// TwinCAT 3 PLC project HD_PLC
// ProgramVersion: 3.1.4024.0
// libraries:
//   Tc2_ModbusRTU, * (Beckhoff Automation GmbH)
//   Tc2_Standard, * (Beckhoff Automation GmbH)
//   Tc2_System, * (Beckhoff Automation GmbH)
//   Tc2_Utilities, * (Beckhoff Automation GmbH)
//   Tc3_Module, * (Beckhoff Automation GmbH)
//   VisuDialogs, * (System)
//   VisuSymbols,3.5.10.0,System
// project tree:
//   / GlobalTextList.TcGTLO, PlcTask.TcTTO, Visualization Manager.TcVMO (not stored), VISU_TASK.TcTTO
//   GVLs/ HMI_Global.TcGVL
//   POUs/ MAIN.TcPOU, SYSTEM.TcPOU
//   VISUs/ Data_Left.TcVIS, Footer.TcVIS, Header.TcVIS, Header_2.TcVIS, ImagePool.TcIPO (not stored), MainScreen.TcVIS, RinseMode.TcVIS, RinseMode_Footer.TcVIS, Set.TcVIS, Set_Output.TcVIS, Set_Input.TcVIS, Set_Sensor.TcVIS, Visualization.TcVIS
// real-time tasks:
//   TASK PlcTask: cycle T#10ms, priority 20, ADS port 350
//   TASK VISU_TASK: cycle T#10ms, priority 1, ADS port 351
//   TASK VISU_TASK1: cycle T#200000us, priority 30, ADS port 352

CONFIGURATION HD_PLC
    RESOURCE PLC ON TwinCAT3
        TASK PlcTask(INTERVAL := T#10ms, PRIORITY := 20);
        TASK VISU_TASK(INTERVAL := T#200000us, PRIORITY := 30);
        PROGRAM MAIN WITH PlcTask : MAIN;
        PROGRAM SYSTEM WITH PlcTask : SYSTEM;
        PROGRAM VisuElems_Visu_Prg WITH VISU_TASK : VisuElems.Visu_Prg;
    END_RESOURCE
END_CONFIGURATION

// ---- GVLs/HMI_Global.TcGVL
{attribute 'qualified_only'}
VAR_GLOBAL
	//HMI Stuff
	HMI_OUT_Digital 	: ARRAY[0..31] OF BOOL;
	HMI_OUT_Analog 		: ARRAY[0..31] OF INT;
	
	HMI_IN_Digital 		: ARRAY[0..31] OF BOOL;
	HMI_IN_Analog 		: ARRAY[0..31] OF INT;
	
	HMI_IN_Temp 		: ARRAY[0..4] OF REAL;
	
	HMI_State			: INT;
	
	fbGetLocalSystemTime: FB_LocalSystemTime;
	sSystemDateTime : STRING;
	sSystemTime		: STRING;
	sSystemDate		: STRING;
	
	HMI_ArrayGraph1 : ARRAY[0..1] OF INT;
	HMI_ArrayGraph2 : ARRAY[0..1] OF INT;
	HMI_ArrayGraph3 : ARRAY[0..1] OF INT;

END_VAR

// ---- POUs/MAIN.TcPOU
PROGRAM MAIN
VAR
	
	CountScale : BYTE;

	Mux_Select AT %Q*: ARRAY[0..4] OF BOOL;	
	ADC_Val AT %I* : INT; 
	AnalogRead : ARRAY[0..31] OF INT;
	CLK_MUX : BOOL;
	
	MUX_FUNC : MUX_ADC;

	IO_Out AT %Q* : ARRAY[0..31] OF BOOL;
	IO_In AT %I* : ARRAY[0..16] OF BOOL;
	
	SensAnalaog AT %I* : ARRAY[0..3] OF INT;
	
	RTD_ADC AT %I* : INT;
	RTD_Temp : REAL;
	
	

END_VAR

CLK_MUX := NOT(CLK_MUX);

IO_Out[8] := HMI_Global.HMI_IN_Digital[0];
HMI_Global.HMI_OUT_Analog[0] := AnalogRead[9];

IF AnalogRead[9] > 1000 THEN
	HMI_Global.HMI_OUT_Digital[0] := TRUE;
ELSE
	HMI_Global.HMI_OUT_Digital[0] := FALSE;
END_IF
 

MUX_FUNC(
	CLK := CLK_MUX,
	ADC_INPUT := ADC_Val,
	SELLECT => Mux_Select,
	ADC_OUTPUT => AnalogRead	
);

END_PROGRAM

// ---- POUs/SYSTEM.TcPOU
PROGRAM SYSTEM
VAR
END_VAR

HMI_Global.fbGetLocalSystemTime(
	sNetID:= , 
	bEnable:= TRUE, 
	dwCycle:= 1, 
	dwOpt:= , 
	tTimeout:= , 
	bValid=> , 
	systemTime=> , 
	tzID=> );
	
HMI_Global.sSystemDateTime := SYSTEMTIME_TO_STRING(HMI_Global.fbGetLocalSystemTime.systemTime);
HMI_Global.sSystemDate := MID(STR:= HMI_Global.sSystemDateTime, LEN:=10, POS:=1);
HMI_Global.sSystemTime := MID(STR:= HMI_Global.sSystemDateTime, LEN:=8, POS:=12);

END_PROGRAM

// ---- GlobalTextList.TcGTLO
TEXTLIST GlobalTextList
  734 = '%1.1f'
  899 = '%2.2f'
  70 = '%i'
  841 = '%s'
  97 = '10'
  56 = '120'
  900 = '30'
  405 = '36'
  563 = '60'
  451 = 'A. PRESS'
  564 = 'B1'
  765 = 'B10'
  285 = 'B11'
  111 = 'B12'
  897 = 'B13'
  671 = 'B14'
  804 = 'B15'
  328 = 'B16'
  300 = 'B17'
  486 = 'B18'
  957 = 'B19'
  273 = 'B2'
  588 = 'B20'
  314 = 'B21'
  91 = 'B22'
  991 = 'B23'
  768 = 'B24'
  634 = 'B25'
  160 = 'B26'
  185 = 'B27'
  572 = 'B28'
  78 = 'B29'
  783 = 'B3'
  964 = 'B30'
  98 = 'B31'
  326 = 'B32'
  703 = 'B4'
  227 = 'B5'
  844 = 'B6'
  235 = 'B7'
  599 = 'B8'
  248 = 'B9'
  100 = 'BACK'
  372 = 'Bic.'
  816 = 'BLOOD PUMP'
  325 = 'Button 1'
  42 = 'Button 2'
  879 = 'Button 3'
  476 = 'Button 4'
  556 = 'Button 5'
  421 = 'Button 6'
  73 = 'Button 7'
  541 = 'Button 8'
  424 = 'Button 9'
  46 = 'BY PAS'
  570 = 'BYPASS'
  2 = 'BYPASS\nRELEASE'
  359 = 'CHECK AND TEST FUNCTION'
  724 = 'CONC. SET'
  918 = 'COND.'
  942 = 'D. PRESS'
  223 = 'DIALYSE'
  633 = 'DIALYSIS'
  645 = 'EST. UF TIME'
  400 = 'HEMODIALYSIS'
  102 = 'HMI STATE'
  583 = 'INPUT'
  17 = 'Input'
  280 = 'Input \nDigital'
  439 = 'Input Digital'
  212 = 'InputDigital'
  770 = 'ISO-UF\n[1sec]'
  733 = 'mmHg'
  339 = 'Na'
  358 = 'NEXT'
  851 = 'ON / OFF'
  71 = 'OUTPUT'
  279 = 'PREP'
  48 = 'PREP. COMP.'
  59 = 'PRIM.'
  370 = 'RINSE\nMODE'
  863 = 'S/N\n[1sec]'
  925 = 'SENSOR'
  498 = 'SET'
  446 = 'TEMP.'
  666 = 'Temperature'
  237 = 'TEST'
  818 = 'UF DATA'
  819 = 'UF FINISH TIME'
  812 = 'UF GOAL'
  795 = 'UF RATE'
  493 = 'UF REMOVED'
  45 = 'V. PRESS'
  944 = '[C]'
  752 = '[h:min]'
  79 = '[L/h]'
  193 = '[L]'
  495 = '[mEq/L]'
  6 = '[mL/min]'
  374 = '[mS/cm]'
END_TEXTLIST

// ---- VISUs/Data_Left.TcVIS
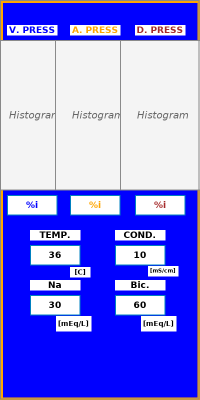
VISUALIZATION Data_Left  // 200x400
    Rectangle (0,0 200x400)
    Histogram (-8,40 86x150), scale format: %1.1f, scale -100..300
        p518627256: mmHg
        p1518820177: HMI_Global.HMI_ArrayGraph1
        p102497268: HMI_Global.HMI_ArrayGraph1
        p788070771: ARRAY [0..1] OF INT
    Histogram (55,40 86x150), scale format: %1.1f, scale -300..100
        p518627256: mmHg
        p1518820177: HMI_Global.HMI_ArrayGraph2
        p102497268: HMI_Global.HMI_ArrayGraph2
        p788070771: ARRAY [0..1] OF INT
    Histogram (120,40 86x150), scale format: %1.1f, scale -400..300
        p518627256: mmHg
        p1518820177: HMI_Global.HMI_ArrayGraph3
        p102497268: HMI_Global.HMI_ArrayGraph3
        p788070771: ARRAY [0..1] OF INT
    Textfield (7,25 50x10), "V. PRESS"
    Textfield (70,25 50x10), "A. PRESS"
    Textfield (135,25 50x10), "D. PRESS"
    Textfield (7,195 50x20), "%i"
    Textfield (70,195 50x20), "%i"
    Textfield (135,195 50x20), "%i"
    Textfield (30,245 50x20), "36"
    Textfield (115,295 50x20), "60"
    Textfield (115,245 50x20), "10"
    Textfield (30,295 50x20), "30"
    Textfield (30,230 50x10), "TEMP."
    Textfield (115,230 50x10), "COND."
    Textfield (115,280 50x10), "Bic."
    Textfield (30,280 50x10), "Na"
    Textfield (70,267 20x10), "[C]"
    Textfield (148,266 30x10), "[mS/cm]"
    Textfield (56,316 35x15), "[mEq/L]"
    Textfield (141,316 35x15), "[mEq/L]"
END_VISUALIZATION

// ---- VISUs/Footer.TcVIS
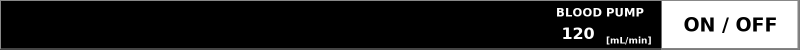
VISUALIZATION Footer  // 800x50
    Rectangle (0,0 800x50)
    Button (661,0 139x50), "ON / OFF"
    Textfield (550,0 100x25), "BLOOD PUMP"
    Textfield (528,21 100x25), "120"
    Textfield (579,28 100x25), "[mL/min]"
END_VISUALIZATION

// ---- VISUs/Header.TcVIS
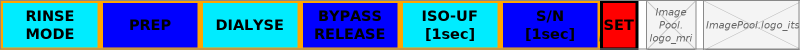
VISUALIZATION Header  // 800x50
    Rectangle (0,0 100x50), "RINSE MODE"
    Rectangle (100,0 100x50), "PREP"
    Rectangle (200,0 100x50), "DIALYSE"
    Rectangle (300,0 100x50), "BYPASS RELEASE", tooltip "BY PAS"
    Rectangle (400,0 100x50), "ISO-UF [1sec]"
    Rectangle (500,0 100x50), "S/N [1sec]"
    Image (600,0 25x50), image: ImagePool.logo_its
    Image (646,0 50x50), image: ImagePool.logo_mri
    Rectangle (600,0 38x50), "SET"
    Image (703,0 100x50), image: ImagePool.logo_its
END_VISUALIZATION

// ---- VISUs/Header_2.TcVIS
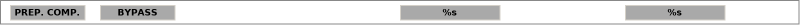
VISUALIZATION Header_2  // 800x25
    Textfield (400,5 75x15), "PREP. COMP."
    Textfield (100,5 75x15), "BYPASS"
    Textfield (400,5 100x15), "%s", text variable: HMI_Global.sSystemDate
    Textfield (625,5 100x15), "%s", text variable: HMI_Global.sSystemTime
    Textfield (10,5 75x15), "PREP. COMP."
END_VISUALIZATION

// ---- VISUs/MainScreen.TcVIS
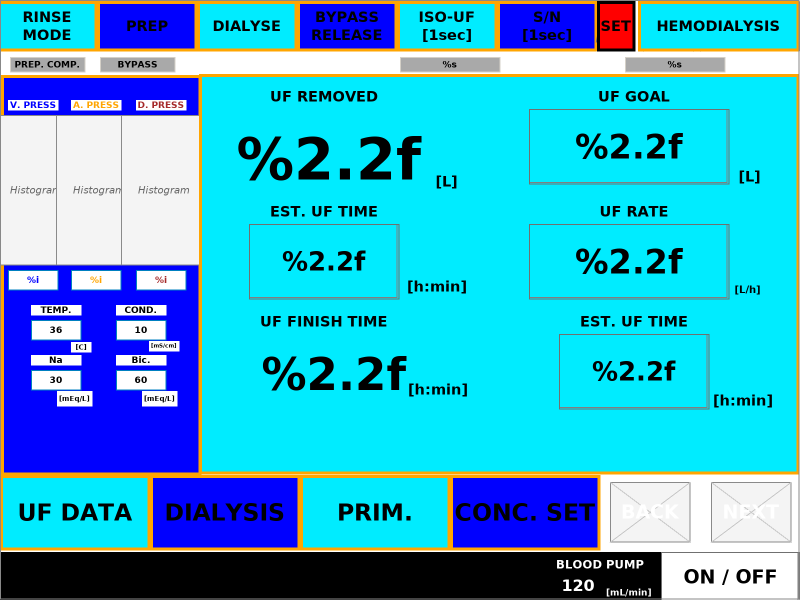
VISUALIZATION MainScreen  // 800x600
    Frame (0,52 800x25)
        shows Header_2()
    Frame (0,552 800x50)
        shows Footer()
    Frame (1,75 200x400)
        shows Data_Left()
    Frame (0,475 800x75)
        shows RinseMode_Footer()
    Rectangle (-3,1 100x50), "RINSE MODE"
        OnMouseClick: FrameSelectionChange Selection=SelectedFrame=2b0ef998-403b-4e78-a897-9d833b853fee, GlobSel=AssignType=Directly, SelType=Locally
    Rectangle (97,1 100x50), "PREP"
    Rectangle (197,1 100x50), "DIALYSE"
    Rectangle (297,1 100x50), "BYPASS RELEASE", tooltip "BY PAS"
    Rectangle (397,1 100x50), "ISO-UF [1sec]"
    Rectangle (497,1 100x50), "S/N [1sec]"
    Image (597,1 25x50), image: ImagePool.logo_its
    Image (643,1 50x50), image: ImagePool.logo_mri
    Rectangle (597,1 38x50), "SET"
        OnMouseClick: FrameSelectionChange Selection=SelectedFrame=2b0ef998-403b-4e78-a897-9d833b853fee, Selection=1, GlobSel=AssignType=Directly, SelType=Locally
    Image (700,1 100x50), image: ImagePool.logo_its
    Frame (199,74 600x400)
        shows RinseMode()
        shows Set()
    Rectangle (638,1 161x50), "HEMODIALYSIS"
END_VISUALIZATION

// ---- VISUs/RinseMode.TcVIS
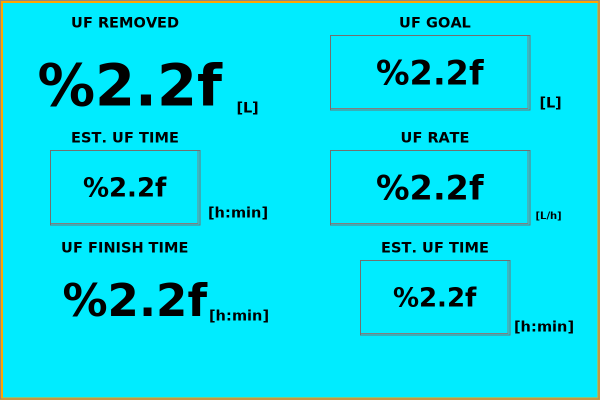
VISUALIZATION RinseMode  // 600x400
    Textfield (0,0 600x400)
    Textfield (50,10 150x25), "UF REMOVED"
    Textfield (360,125 150x25), "UF RATE"
    Textfield (5,35 250x100), "%2.2f"
    Button (330,35 200x75), "%2.2f"
        OnMouseDown: write the text variable via VisuDialogs.Numpad, min 0, max 1000
    Textfield (360,10 150x25), "UF GOAL"
    Button (330,150 200x75), "%2.2f"
        OnMouseDown: write the text variable via VisuDialogs.Numpad, min 0, max 1000
    Button (50,150 150x75), "%2.2f"
        OnMouseDown: write the text variable via VisuDialogs.Numpad, min 0, max 1000
    Textfield (50,125 150x25), "EST. UF TIME"
    Textfield (779,143 1x0)
    Textfield (536,203 25x25), "[L/h]"
    Textfield (538,90 25x25), "[L]"
    Textfield (235,95 25x25), "[L]"
    Textfield (206,200 64x25), "[h:min]"
    Button (360,260 150x75), "%2.2f"
        OnMouseDown: write the text variable via VisuDialogs.Numpad, min 0, max 1000
    Textfield (360,235 150x25), "EST. UF TIME"
    Textfield (512,314 64x25), "[h:min]"
    Textfield (10,250 250x100), "%2.2f"
    Textfield (50,235 150x25), "UF FINISH TIME"
    Textfield (207,303 64x25), "[h:min]"
END_VISUALIZATION

// ---- VISUs/RinseMode_Footer.TcVIS
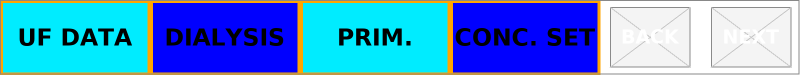
VISUALIZATION RinseMode_Footer  // 800x75
    Textfield (0,0 150x75), "UF DATA"
    Textfield (150,0 150x75), "DIALYSIS"
    Textfield (300,0 150x75), "PRIM."
    Textfield (450,0 150x75), "CONC. SET"
    Image (610,7 80x60), "BACK", image: VisuSymbols.Symbols.ArrowBoldLeft
    Image (711,7 80x60), "NEXT", image: VisuSymbols.Symbols.ArrowBoldRight
END_VISUALIZATION

// ---- VISUs/Set.TcVIS
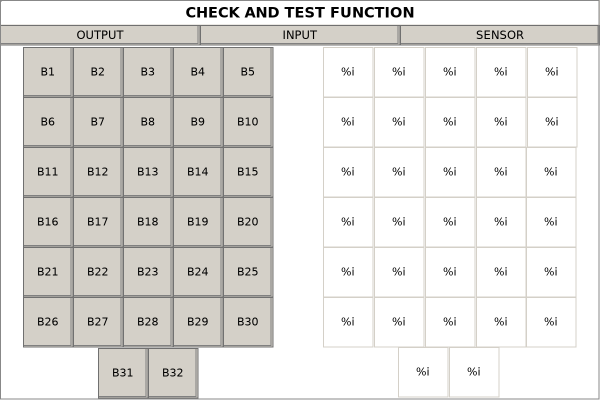
VISUALIZATION Set  // 600x400
    Textfield (0,0 600x25), "CHECK AND TEST FUNCTION"
    Rectangle (0,0 1x0)
    Frame (3,45 600x355)
        shows Set_Output()
        shows Set_Input()
        shows Set_Sensor()
    Button (0,25 200x20), "OUTPUT"
        OnMouseClick: FrameSelectionChange Selection=SelectedFrame=0fef5f47-d526-41e0-bfa2-b91095b14cc7, GlobSel=AssignType=Directly, SelType=Locally
    Button (400,25 200x20), "SENSOR"
        OnMouseClick: FrameSelectionChange Selection=SelectedFrame=0fef5f47-d526-41e0-bfa2-b91095b14cc7, Selection=2, GlobSel=AssignType=Directly, SelType=Locally
    Button (200,25 200x20), "INPUT"
        OnMouseClick: FrameSelectionChange Selection=SelectedFrame=0fef5f47-d526-41e0-bfa2-b91095b14cc7, Selection=1, GlobSel=AssignType=Directly, SelType=Locally
END_VISUALIZATION

// ---- VISUs/Set_Output.TcVIS
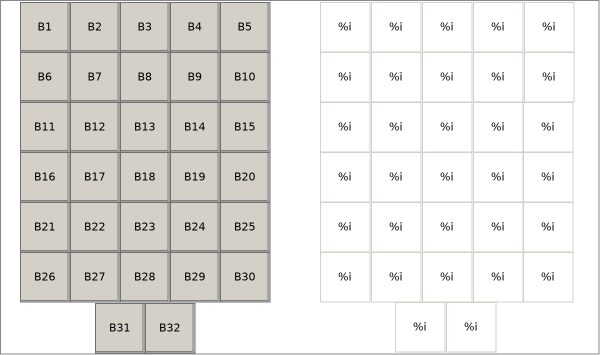
VISUALIZATION Set_Output  // 600x355
    Button (20,2 50x50), "B1", colour toggle: HMI_Global.HMI_OUT_Digital[0]
        toggle HMI_Global.HMI_OUT_Digital[0]
    Textfield (320,2 50x50), "%i", text variable: HMI_Global.HMI_OUT_Analog[0]
        OnMouseDown: write the text variable via VisuDialogs.Numpad, min 0, max 1000
    Button (70,2 50x50), "B2", colour toggle: HMI_Global.HMI_OUT_Digital[1]
        toggle HMI_Global.HMI_OUT_Digital[1]
    Button (120,2 50x50), "B3", colour toggle: HMI_Global.HMI_OUT_Digital[2]
        toggle HMI_Global.HMI_OUT_Digital[2]
    Button (170,2 50x50), "B4", colour toggle: HMI_Global.HMI_OUT_Digital[3]
        toggle HMI_Global.HMI_OUT_Digital[3]
    Button (220,2 50x50), "B5", colour toggle: HMI_Global.HMI_OUT_Digital[4]
        toggle HMI_Global.HMI_OUT_Digital[4]
    Button (20,52 50x50), "B6", colour toggle: HMI_Global.HMI_OUT_Digital[5]
        toggle HMI_Global.HMI_OUT_Digital[5]
    Button (70,52 50x50), "B7", colour toggle: HMI_Global.HMI_OUT_Digital[6]
        toggle HMI_Global.HMI_OUT_Digital[6]
    Button (120,52 50x50), "B8", colour toggle: HMI_Global.HMI_OUT_Digital[7]
        toggle HMI_Global.HMI_OUT_Digital[7]
    Button (170,52 50x50), "B9", colour toggle: HMI_Global.HMI_OUT_Digital[8]
        toggle HMI_Global.HMI_OUT_Digital[8]
    Button (220,52 50x50), "B10", colour toggle: HMI_Global.HMI_OUT_Digital[9]
        toggle HMI_Global.HMI_OUT_Digital[9]
    Button (20,152 50x50), "B16", colour toggle: HMI_Global.HMI_OUT_Digital[15]
        toggle HMI_Global.HMI_OUT_Digital[15]
    Button (20,102 50x50), "B11", colour toggle: HMI_Global.HMI_OUT_Digital[10]
        toggle HMI_Global.HMI_OUT_Digital[10]
    Button (70,102 50x50), "B12", colour toggle: HMI_Global.HMI_OUT_Digital[11]
        toggle HMI_Global.HMI_OUT_Digital[11]
    Button (120,102 50x50), "B13", colour toggle: HMI_Global.HMI_OUT_Digital[12]
        toggle HMI_Global.HMI_OUT_Digital[12]
    Button (170,102 50x50), "B14", colour toggle: HMI_Global.HMI_OUT_Digital[13]
        toggle HMI_Global.HMI_OUT_Digital[13]
    Button (220,102 50x50), "B15", colour toggle: HMI_Global.HMI_OUT_Digital[14]
        toggle HMI_Global.HMI_OUT_Digital[14]
    Button (70,152 50x50), "B17", colour toggle: HMI_Global.HMI_OUT_Digital[16]
        toggle HMI_Global.HMI_OUT_Digital[16]
    Button (120,152 50x50), "B18", colour toggle: HMI_Global.HMI_OUT_Digital[17]
        toggle HMI_Global.HMI_OUT_Digital[17]
    Button (170,152 50x50), "B19", colour toggle: HMI_Global.HMI_OUT_Digital[18]
        toggle HMI_Global.HMI_OUT_Digital[18]
    Button (220,152 50x50), "B20", colour toggle: HMI_Global.HMI_OUT_Digital[19]
        toggle HMI_Global.HMI_OUT_Digital[19]
    Button (20,202 50x50), "B21", colour toggle: HMI_Global.HMI_OUT_Digital[20]
        toggle HMI_Global.HMI_OUT_Digital[20]
    Button (20,252 50x50), "B26", colour toggle: HMI_Global.HMI_OUT_Digital[25]
        toggle HMI_Global.HMI_OUT_Digital[25]
    Button (70,202 50x50), "B22", colour toggle: HMI_Global.HMI_OUT_Digital[21]
        toggle HMI_Global.HMI_OUT_Digital[21]
    Button (120,202 50x50), "B23", colour toggle: HMI_Global.HMI_OUT_Digital[22]
        toggle HMI_Global.HMI_OUT_Digital[22]
    Button (170,202 50x50), "B24", colour toggle: HMI_Global.HMI_OUT_Digital[23]
        toggle HMI_Global.HMI_OUT_Digital[23]
    Button (220,202 50x50), "B25", colour toggle: HMI_Global.HMI_OUT_Digital[24]
        toggle HMI_Global.HMI_OUT_Digital[24]
    Button (70,252 50x50), "B27", colour toggle: HMI_Global.HMI_OUT_Digital[26]
        toggle HMI_Global.HMI_OUT_Digital[26]
    Button (120,252 50x50), "B28", colour toggle: HMI_Global.HMI_OUT_Digital[27]
        toggle HMI_Global.HMI_OUT_Digital[27]
    Button (170,252 50x50), "B29", colour toggle: HMI_Global.HMI_OUT_Digital[28]
        toggle HMI_Global.HMI_OUT_Digital[28]
    Button (220,252 50x50), "B30", colour toggle: HMI_Global.HMI_OUT_Digital[29]
        toggle HMI_Global.HMI_OUT_Digital[29]
    Button (95,303 50x50), "B31", colour toggle: HMI_Global.HMI_OUT_Digital[30]
        toggle HMI_Global.HMI_OUT_Digital[30]
    Button (145,303 50x50), "B32", colour toggle: HMI_Global.HMI_OUT_Digital[31]
        toggle HMI_Global.HMI_OUT_Digital[31]
    Textfield (371,2 50x50), "%i", text variable: HMI_Global.HMI_OUT_Analog[1]
        OnMouseDown: write the text variable via VisuDialogs.Numpad, min 0, max 1000
    Textfield (422,2 50x50), "%i", text variable: HMI_Global.HMI_OUT_Analog[2]
        OnMouseDown: write the text variable via VisuDialogs.Numpad, min 0, max 1000
    Textfield (473,2 50x50), "%i", text variable: HMI_Global.HMI_OUT_Analog[3]
        OnMouseDown: write the text variable via VisuDialogs.Numpad, min 0, max 1000
    Textfield (524,2 50x50), "%i", text variable: HMI_Global.HMI_OUT_Analog[4]
        OnMouseDown: write the text variable via VisuDialogs.Numpad, min 0, max 1000
    Textfield (320,52 50x50), "%i", text variable: HMI_Global.HMI_OUT_Analog[5]
        OnMouseDown: write the text variable via VisuDialogs.Numpad, min 0, max 1000
    Textfield (371,52 50x50), "%i", text variable: HMI_Global.HMI_OUT_Analog[6]
        OnMouseDown: write the text variable via VisuDialogs.Numpad, min 0, max 1000
    Textfield (422,52 50x50), "%i", text variable: HMI_Global.HMI_OUT_Analog[7]
        OnMouseDown: write the text variable via VisuDialogs.Numpad, min 0, max 1000
    Textfield (473,52 50x50), "%i", text variable: HMI_Global.HMI_OUT_Analog[8]
        OnMouseDown: write the text variable via VisuDialogs.Numpad, min 0, max 1000
    Textfield (524,52 50x50), "%i", text variable: HMI_Global.HMI_OUT_Analog[9]
        OnMouseDown: write the text variable via VisuDialogs.Numpad, min 0, max 1000
    Textfield (320,102 50x50), "%i", text variable: HMI_Global.HMI_OUT_Analog[10]
        OnMouseDown: write the text variable via VisuDialogs.Numpad, min 0, max 1000
    Textfield (371,102 50x50), "%i", text variable: HMI_Global.HMI_OUT_Analog[11]
        OnMouseDown: write the text variable via VisuDialogs.Numpad, min 0, max 1000
    Textfield (422,102 50x50), "%i", text variable: HMI_Global.HMI_OUT_Analog[12]
        OnMouseDown: write the text variable via VisuDialogs.Numpad, min 0, max 1000
    Textfield (473,102 50x50), "%i", text variable: HMI_Global.HMI_OUT_Analog[13]
        OnMouseDown: write the text variable via VisuDialogs.Numpad, min 0, max 1000
    Textfield (523,102 50x50), "%i", text variable: HMI_Global.HMI_OUT_Analog[14]
        OnMouseDown: write the text variable via VisuDialogs.Numpad, min 0, max 1000
    Textfield (320,152 50x50), "%i", text variable: HMI_Global.HMI_OUT_Analog[15]
        OnMouseDown: write the text variable via VisuDialogs.Numpad, min 0, max 1000
    Textfield (371,152 50x50), "%i", text variable: HMI_Global.HMI_OUT_Analog[16]
        OnMouseDown: write the text variable via VisuDialogs.Numpad, min 0, max 1000
    Textfield (422,152 50x50), "%i", text variable: HMI_Global.HMI_OUT_Analog[17]
        OnMouseDown: write the text variable via VisuDialogs.Numpad, min 0, max 1000
    Textfield (473,152 50x50), "%i", text variable: HMI_Global.HMI_OUT_Analog[18]
        OnMouseDown: write the text variable via VisuDialogs.Numpad, min 0, max 1000
    Textfield (523,152 50x50), "%i", text variable: HMI_Global.HMI_OUT_Analog[19]
        OnMouseDown: write the text variable via VisuDialogs.Numpad, min 0, max 1000
    Textfield (320,202 50x50), "%i", text variable: HMI_Global.HMI_OUT_Analog[20]
        OnMouseDown: write the text variable via VisuDialogs.Numpad, min 0, max 1000
    Textfield (371,202 50x50), "%i", text variable: HMI_Global.HMI_OUT_Analog[21]
        OnMouseDown: write the text variable via VisuDialogs.Numpad, min 0, max 1000
    Textfield (422,202 50x50), "%i", text variable: HMI_Global.HMI_OUT_Analog[22]
        OnMouseDown: write the text variable via VisuDialogs.Numpad, min 0, max 1000
    Textfield (473,202 50x50), "%i", text variable: HMI_Global.HMI_OUT_Analog[23]
        OnMouseDown: write the text variable via VisuDialogs.Numpad, min 0, max 1000
    Textfield (523,202 50x50), "%i", text variable: HMI_Global.HMI_OUT_Analog[24]
        OnMouseDown: write the text variable via VisuDialogs.Numpad, min 0, max 1000
    Textfield (320,252 50x50), "%i", text variable: HMI_Global.HMI_OUT_Analog[25]
        OnMouseDown: write the text variable via VisuDialogs.Numpad, min 0, max 1000
    Textfield (371,252 50x50), "%i", text variable: HMI_Global.HMI_OUT_Analog[26]
        OnMouseDown: write the text variable via VisuDialogs.Numpad, min 0, max 1000
    Textfield (422,252 50x50), "%i", text variable: HMI_Global.HMI_OUT_Analog[27]
        OnMouseDown: write the text variable via VisuDialogs.Numpad, min 0, max 1000
    Textfield (473,252 50x50), "%i", text variable: HMI_Global.HMI_OUT_Analog[28]
        OnMouseDown: write the text variable via VisuDialogs.Numpad, min 0, max 1000
    Textfield (523,252 50x50), "%i", text variable: HMI_Global.HMI_OUT_Analog[29]
        OnMouseDown: write the text variable via VisuDialogs.Numpad, min 0, max 1000
    Textfield (395,302 50x50), "%i", text variable: HMI_Global.HMI_OUT_Analog[30]
        OnMouseDown: write the text variable via VisuDialogs.Numpad, min 0, max 1000
    Textfield (446,302 50x50), "%i", text variable: HMI_Global.HMI_OUT_Analog[31]
        OnMouseDown: write the text variable via VisuDialogs.Numpad, min 0, max 1000
END_VISUALIZATION

// ---- VISUs/Set_Input.TcVIS
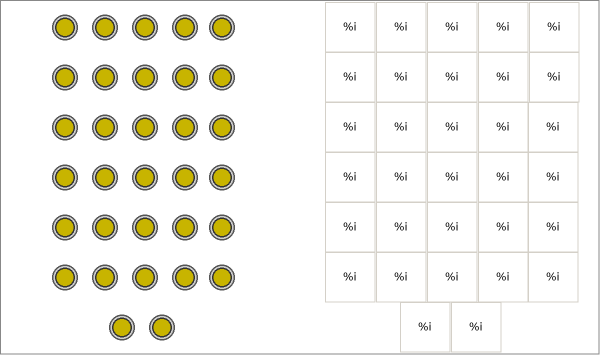
VISUALIZATION Set_Input  // 600x355
    Lamp1 (50,10 30x35), variable: HMI_Global.HMI_IN_Digital[0], style: Lamp-Lamp1-Yellow
    Lamp1 (90,10 30x35), variable: HMI_Global.HMI_IN_Digital[1], style: Lamp-Lamp1-Yellow
    Lamp1 (130,10 30x35), variable: HMI_Global.HMI_IN_Digital[2], style: Lamp-Lamp1-Yellow
    Lamp1 (170,10 30x35), variable: HMI_Global.HMI_IN_Digital[3], style: Lamp-Lamp1-Yellow
    Lamp1 (170,60 30x35), variable: HMI_Global.HMI_IN_Digital[8], style: Lamp-Lamp1-Yellow
    Lamp1 (50,60 30x35), variable: HMI_Global.HMI_IN_Digital[5], style: Lamp-Lamp1-Yellow
    Lamp1 (90,60 30x35), variable: HMI_Global.HMI_IN_Digital[6], style: Lamp-Lamp1-Yellow
    Lamp1 (130,60 30x35), variable: HMI_Global.HMI_IN_Digital[7], style: Lamp-Lamp1-Yellow
    Lamp1 (50,110 30x35), variable: HMI_Global.HMI_IN_Digital[10], style: Lamp-Lamp1-Yellow
    Lamp1 (170,110 30x35), variable: HMI_Global.HMI_IN_Digital[13], style: Lamp-Lamp1-Yellow
    Lamp1 (90,110 30x35), variable: HMI_Global.HMI_IN_Digital[11], style: Lamp-Lamp1-Yellow
    Lamp1 (130,110 30x35), variable: HMI_Global.HMI_IN_Digital[12], style: Lamp-Lamp1-Yellow
    Lamp1 (50,160 30x35), variable: HMI_Global.HMI_IN_Digital[15], style: Lamp-Lamp1-Yellow
    Lamp1 (90,160 30x35), variable: HMI_Global.HMI_IN_Digital[16], style: Lamp-Lamp1-Yellow
    Lamp1 (130,160 30x35), variable: HMI_Global.HMI_IN_Digital[17], style: Lamp-Lamp1-Yellow
    Lamp1 (170,160 30x35), variable: HMI_Global.HMI_IN_Digital[18], style: Lamp-Lamp1-Yellow
    Lamp1 (170,210 30x35), variable: HMI_Global.HMI_IN_Digital[23], style: Lamp-Lamp1-Yellow
    Lamp1 (50,210 30x35), variable: HMI_Global.HMI_IN_Digital[20], style: Lamp-Lamp1-Yellow
    Lamp1 (90,210 30x35), variable: HMI_Global.HMI_IN_Digital[21], style: Lamp-Lamp1-Yellow
    Lamp1 (130,210 30x35), variable: HMI_Global.HMI_IN_Digital[22], style: Lamp-Lamp1-Yellow
    Lamp1 (207,10 30x35), variable: HMI_Global.HMI_IN_Digital[4], style: Lamp-Lamp1-Yellow
    Lamp1 (207,60 30x35), variable: HMI_Global.HMI_IN_Digital[9], style: Lamp-Lamp1-Yellow
    Lamp1 (207,110 30x35), variable: HMI_Global.HMI_IN_Digital[14], style: Lamp-Lamp1-Yellow
    Lamp1 (207,160 30x35), variable: HMI_Global.HMI_IN_Digital[19], style: Lamp-Lamp1-Yellow
    Lamp1 (207,210 30x35), variable: HMI_Global.HMI_IN_Digital[24], style: Lamp-Lamp1-Yellow
    Lamp1 (170,260 30x35), variable: HMI_Global.HMI_IN_Digital[28], style: Lamp-Lamp1-Yellow
    Lamp1 (50,260 30x35), variable: HMI_Global.HMI_IN_Digital[25], style: Lamp-Lamp1-Yellow
    Lamp1 (90,260 30x35), variable: HMI_Global.HMI_IN_Digital[26], style: Lamp-Lamp1-Yellow
    Lamp1 (130,260 30x35), variable: HMI_Global.HMI_IN_Digital[27], style: Lamp-Lamp1-Yellow
    Lamp1 (207,260 30x35), variable: HMI_Global.HMI_IN_Digital[29], style: Lamp-Lamp1-Yellow
    Textfield (325,2 50x50), "%i", text variable: HMI_Global.HMI_IN_Analog[0]
        OnMouseDown: write the text variable via VisuDialogs.Numpad, min 0, max 1000
    Textfield (376,2 50x50), "%i", text variable: HMI_Global.HMI_IN_Analog[1]
        OnMouseDown: write the text variable via VisuDialogs.Numpad, min 0, max 1000
    Textfield (427,2 50x50), "%i", text variable: HMI_Global.HMI_IN_Analog[2]
        OnMouseDown: write the text variable via VisuDialogs.Numpad, min 0, max 1000
    Textfield (478,2 50x50), "%i", text variable: HMI_Global.HMI_IN_Analog[3]
        OnMouseDown: write the text variable via VisuDialogs.Numpad, min 0, max 1000
    Textfield (529,2 50x50), "%i", text variable: HMI_Global.HMI_IN_Analog[4]
        OnMouseDown: write the text variable via VisuDialogs.Numpad, min 0, max 1000
    Textfield (325,52 50x50), "%i", text variable: HMI_Global.HMI_IN_Analog[5]
        OnMouseDown: write the text variable via VisuDialogs.Numpad, min 0, max 1000
    Textfield (376,52 50x50), "%i", text variable: HMI_Global.HMI_IN_Analog[6]
        OnMouseDown: write the text variable via VisuDialogs.Numpad, min 0, max 1000
    Textfield (427,52 50x50), "%i", text variable: HMI_Global.HMI_IN_Analog[7]
        OnMouseDown: write the text variable via VisuDialogs.Numpad, min 0, max 1000
    Textfield (478,52 50x50), "%i", text variable: HMI_Global.HMI_IN_Analog[8]
        OnMouseDown: write the text variable via VisuDialogs.Numpad, min 0, max 1000
    Textfield (529,52 50x50), "%i", text variable: HMI_Global.HMI_IN_Analog[9]
        OnMouseDown: write the text variable via VisuDialogs.Numpad, min 0, max 1000
    Textfield (325,102 50x50), "%i", text variable: HMI_Global.HMI_IN_Analog[10]
        OnMouseDown: write the text variable via VisuDialogs.Numpad, min 0, max 1000
    Textfield (376,102 50x50), "%i", text variable: HMI_Global.HMI_IN_Analog[11]
        OnMouseDown: write the text variable via VisuDialogs.Numpad, min 0, max 1000
    Textfield (427,102 50x50), "%i", text variable: HMI_Global.HMI_IN_Analog[12]
        OnMouseDown: write the text variable via VisuDialogs.Numpad, min 0, max 1000
    Textfield (478,102 50x50), "%i", text variable: HMI_Global.HMI_IN_Analog[13]
        OnMouseDown: write the text variable via VisuDialogs.Numpad, min 0, max 1000
    Textfield (528,102 50x50), "%i", text variable: HMI_Global.HMI_IN_Analog[14]
        OnMouseDown: write the text variable via VisuDialogs.Numpad, min 0, max 1000
    Textfield (325,152 50x50), "%i", text variable: HMI_Global.HMI_IN_Analog[15]
        OnMouseDown: write the text variable via VisuDialogs.Numpad, min 0, max 1000
    Textfield (376,152 50x50), "%i", text variable: HMI_Global.HMI_IN_Analog[16]
        OnMouseDown: write the text variable via VisuDialogs.Numpad, min 0, max 1000
    Textfield (427,152 50x50), "%i", text variable: HMI_Global.HMI_IN_Analog[17]
        OnMouseDown: write the text variable via VisuDialogs.Numpad, min 0, max 1000
    Textfield (478,152 50x50), "%i", text variable: HMI_Global.HMI_IN_Analog[18]
        OnMouseDown: write the text variable via VisuDialogs.Numpad, min 0, max 1000
    Textfield (528,152 50x50), "%i", text variable: HMI_Global.HMI_IN_Analog[19]
        OnMouseDown: write the text variable via VisuDialogs.Numpad, min 0, max 1000
    Textfield (325,202 50x50), "%i", text variable: HMI_Global.HMI_IN_Analog[20]
        OnMouseDown: write the text variable via VisuDialogs.Numpad, min 0, max 1000
    Textfield (376,202 50x50), "%i", text variable: HMI_Global.HMI_IN_Analog[21]
        OnMouseDown: write the text variable via VisuDialogs.Numpad, min 0, max 1000
    Textfield (427,202 50x50), "%i", text variable: HMI_Global.HMI_IN_Analog[22]
        OnMouseDown: write the text variable via VisuDialogs.Numpad, min 0, max 1000
    Textfield (478,202 50x50), "%i", text variable: HMI_Global.HMI_IN_Analog[23]
        OnMouseDown: write the text variable via VisuDialogs.Numpad, min 0, max 1000
    Textfield (528,202 50x50), "%i", text variable: HMI_Global.HMI_IN_Analog[24]
        OnMouseDown: write the text variable via VisuDialogs.Numpad, min 0, max 1000
    Textfield (325,252 50x50), "%i", text variable: HMI_Global.HMI_IN_Analog[25]
        OnMouseDown: write the text variable via VisuDialogs.Numpad, min 0, max 1000
    Textfield (376,252 50x50), "%i", text variable: HMI_Global.HMI_IN_Analog[26]
        OnMouseDown: write the text variable via VisuDialogs.Numpad, min 0, max 1000
    Textfield (427,252 50x50), "%i", text variable: HMI_Global.HMI_IN_Analog[27]
        OnMouseDown: write the text variable via VisuDialogs.Numpad, min 0, max 1000
    Textfield (478,252 50x50), "%i", text variable: HMI_Global.HMI_IN_Analog[28]
        OnMouseDown: write the text variable via VisuDialogs.Numpad, min 0, max 1000
    Textfield (528,252 50x50), "%i", text variable: HMI_Global.HMI_IN_Analog[29]
        OnMouseDown: write the text variable via VisuDialogs.Numpad, min 0, max 1000
    Textfield (400,302 50x50), "%i", text variable: HMI_Global.HMI_IN_Analog[30]
        OnMouseDown: write the text variable via VisuDialogs.Numpad, min 0, max 1000
    Textfield (451,302 50x50), "%i", text variable: HMI_Global.HMI_IN_Analog[31]
        OnMouseDown: write the text variable via VisuDialogs.Numpad, min 0, max 1000
    Lamp1 (107,310 30x35), variable: HMI_Global.HMI_IN_Digital[30], style: Lamp-Lamp1-Yellow
    Lamp1 (147,310 30x35), variable: HMI_Global.HMI_IN_Digital[31], style: Lamp-Lamp1-Yellow
END_VISUALIZATION

// ---- VISUs/Set_Sensor.TcVIS
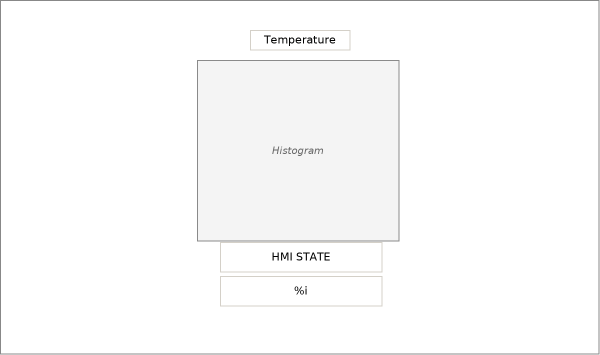
VISUALIZATION Set_Sensor  // 600x355
    Textfield (250,30 100x20), "Temperature"
    Textfield (220,242 162x30), "HMI STATE"
    Textfield (220,276 162x30), "%i", text variable: HMI_Global.HMI_State
    Histogram (197,60 202x181), scale format: %.1f, scale 0..100
        p1518820177: HMI_Global.HMI_IN_Temp
        p102497268: HMI_Global.HMI_IN_Temp
        p788070771: ARRAY [0..4] OF REAL
END_VISUALIZATION

// ---- VISUs/Visualization.TcVIS
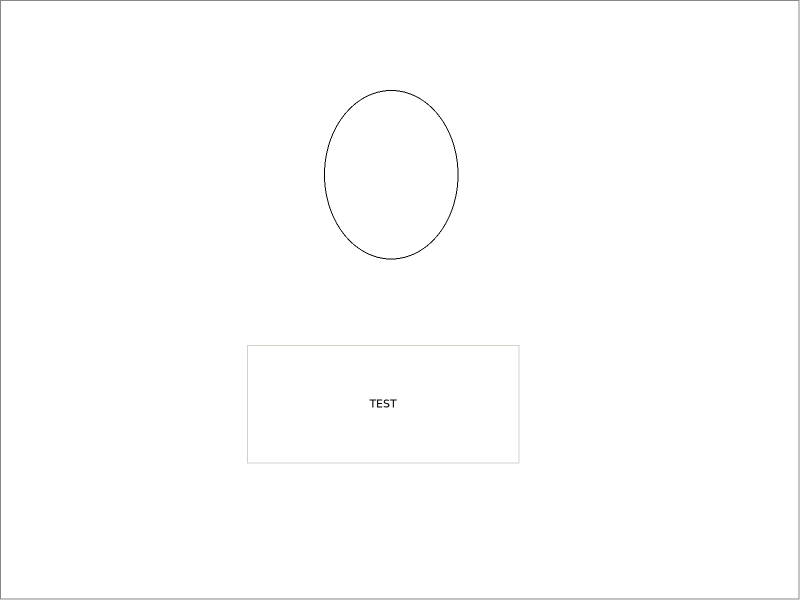
VISUALIZATION Visualization  // 800x600
    Ellipse (324,90 134x169)
    Textfield (247,345 272x118), "TEST"
END_VISUALIZATION
